TYPE Part :
STRUCT
		sn 						: WORD := 0;
		sta1_del 				: ExpTime;
		sta2_del 				: ExpTime;
		sta3_del 				: ExpTime;
		sta4_del 				: ExpTime;
		sta6_del 				: ExpTime;
		sta1_to_sta2_del 		: ExpTime;
		sta2_to_sta3_del 		: ExpTime;
		sta3_to_sta4_del 		: ExpTime;
		sta6_to_sta1_del 		: ExpTime;
		inspection				: WORD := 0;
END_STRUCT
END_TYPE

(* stored: Version 1.1.0.1, ProductVersion 3.1.0.36
   DUT Part: Id {69cfe8f7-6820-4fe4-b464-8d8f862b3056} *)
